(* PLC project VGP - Station 1, CCRE VGP 1.0 *)
(* stored: creationDateTime 2016-05-18T12:27:41, modificationDateTime 2020-06-25T10:53:04 *)

FUNCTION Convert_Pressure : BOOL
  VAR_INPUT
    rawPressure : INT;
  END_VAR
  VAR_OUTPUT
    finalPressure : REAL;
  END_VAR

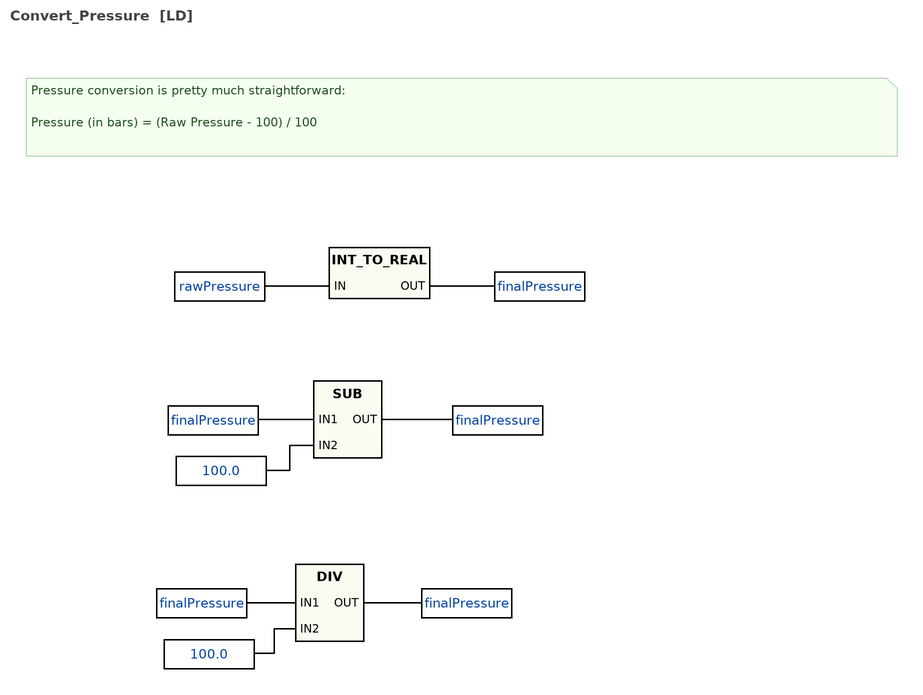
(* LD diagram, written out as Structured Text *)
(* Pressure conversion is pretty much straightforward:

Pressure (in bars) = (Raw Pressure - 100) / 100 *)
finalPressure := INT_TO_REAL(rawPressure);
finalPressure := finalPressure - 100.0;
finalPressure := finalPressure / 100.0;
END_FUNCTION

FUNCTION Finish_Intermediate_Mode : BOOL
  VAR_INPUT
    flow_rate1 : INT;
    flow_rate2 : INT;
    flow_limit : INT;
  END_VAR
  VAR
    negative_flow_limit : INT;
  END_VAR
  VAR_OUTPUT
    Q : BOOL;
  END_VAR

negative_flow_limit := 0 - flow_limit;

IF (negative_flow_limit < flow_rate1) AND (flow_rate1 < flow_limit) THEN
  IF (negative_flow_limit < flow_rate2) AND (flow_rate2 < flow_limit) THEN
    Q := TRUE;
  ELSE
    Q := FALSE;
  END_IF;
ELSE
  Q := FALSE;
END_IF;
          
END_FUNCTION

FUNCTION_BLOCK Verify_Mode_Change
  VAR_INPUT
    mode : INT;
  END_VAR
  VAR_OUTPUT
    Q : BOOL;
  END_VAR
  VAR
    previous_mode : INT := 0;
  END_VAR

IF mode <> previous_mode THEN
  IF (mode > 0) AND (previous_mode > 0) THEN
    Q := TRUE;
  ELSE
    Q := FALSE;
  END_IF;
ELSE
  Q := FALSE;
END_IF;

previous_mode := mode;
          
END_FUNCTION_BLOCK

PROGRAM VGP
  VAR
    raw_pressure AT %IW0 : INT;  (* MODBUS Input Register Address 0 - Pressure as seen from the sensor *)
    raw_tank_lvl AT %IW1 : INT;  (* MODBUS Input Register Address 1 - Tank level as seen from the sensor *)
    raw_dispatch_flow AT %IW2 : INT;  (* MODBUS Input Register Address 2 - Flow rate on the dispatch valve as seen from the sensor *)
    raw_returnline_flow AT %IW3 : INT;  (* MODBUS Input Register Address 3 - Flow rate on the return line as seen from the sensor *)
    raw_relief_valve_flow AT %IW4 : INT;  (* MODBUS Input Register Address 4 - Flow rate on the relief valve as seen from the sensor *)
    raw_min_sp AT %QW1 : INT;  (* MODBUS Holding Register Address 1 - Minimum setpoint (as integer, withouth conversion) *)
    raw_max_sp AT %QW2 : INT;  (* MODBUS Holding Register Address 2 - Maximum setpoint (as integer, withouth conversion) *)
    operation_mode AT %QW3 : INT;  (* MODBUS Holding Register Address 3 - Operation mode, set by the HMI *)
    manual_pump AT %QW4 : INT;  (* MODBUS Holding Register Address 4 - Toggle pump in manual mode *)
    manual_relief_valve AT %QW5 : INT;  (* MODBUS Holding Register Address 5 - Toggle relief valve in manual mode *)
    manual_dispatch_valve AT %QW6 : INT;  (* MODBUS Holding Register Address 6 - Toggle dispatch valve in manual mode *)
    manual_return_valve AT %QW7 : INT;  (* MODBUS Holding Register Address 7 - Toggle return valve in manual mode *)
    source_tank_flow AT %QW20 : INT;  (* MODBUS Holding Register Address 20 - Source Tank flow rate in KL/h *)
    destination_tank_flow AT %QW21 : INT;  (* MODBUS Holding Register Address 21 - Destination Tank flow rate in KL/h *)
    pump AT %QX0.0 : BOOL;
    dispatch_valve AT %QX0.2 : BOOL;
    return_valve AT %QX0.3 : BOOL;
    relief_valve AT %QX0.1 : BOOL;
  END_VAR
  VAR
    pressure : REAL;
    min_sp : REAL;
    max_sp : REAL;
    recirc_mode : BOOL;
    recirc_dispatch_valve : BOOL;
    recirc_return_valve : BOOL;
    recirc_relief_valve : BOOL;
    recirc_pump : BOOL;
    cargo_mode : BOOL;
    cargo_dispatch_valve : BOOL;
    cargo_return_valve : BOOL;
    cargo_relief_valve : BOOL;
    cargo_pump : BOOL;
    man_mode : BOOL;
    man_dispatch_valve : BOOL;
    man_return_valve : BOOL;
    man_relief_valve : BOOL;
    man_pump : BOOL;
    intermediate_mode : BOOL;
    intermediate_dispatch_valve : BOOL;
    intermediate_return_valve : BOOL;
    intermediate_relief_valve : BOOL;
    intermediate_pump : BOOL;
    TOF0 : TOF;
    mode_change : Verify_Mode_Change;
    T0 : TON;
  END_VAR
  VAR  (* added by the conversion: wires and edge detectors of the diagram *)
    _Convert_Pressure152_finalPressure : ANY;
    _Convert_Pressure152_OUT : BOOL;
    _Convert_Pressure153_finalPressure : ANY;
    _Convert_Pressure153_OUT : BOOL;
    _Convert_Pressure154_finalPressure : ANY;
    _Convert_Pressure154_OUT : BOOL;
    _Finish_Intermediate_Mode215_Q : ANY;
    _Finish_Intermediate_Mode215_OUT : BOOL;
    _LE164_ENO : BOOL;
    _LE164_OUT : BOOL;
    _GE169_ENO : BOOL;
    _GE169_OUT : BOOL;
    _GE173_ENO : BOOL;
    _GE173_OUT : BOOL;
    _LE33_ENO : BOOL;
    _LE33_OUT : BOOL;
    _GE38_ENO : BOOL;
    _GE38_OUT : BOOL;
    _EQ42_OUT : BOOL;
    _EQ183_ENO : BOOL;
    _EQ183_OUT : BOOL;
    _EQ49_ENO : BOOL;
    _EQ49_OUT : BOOL;
    _EQ56_ENO : BOOL;
    _EQ56_OUT : BOOL;
    _EQ63_ENO : BOOL;
    _EQ63_OUT : BOOL;
  END_VAR

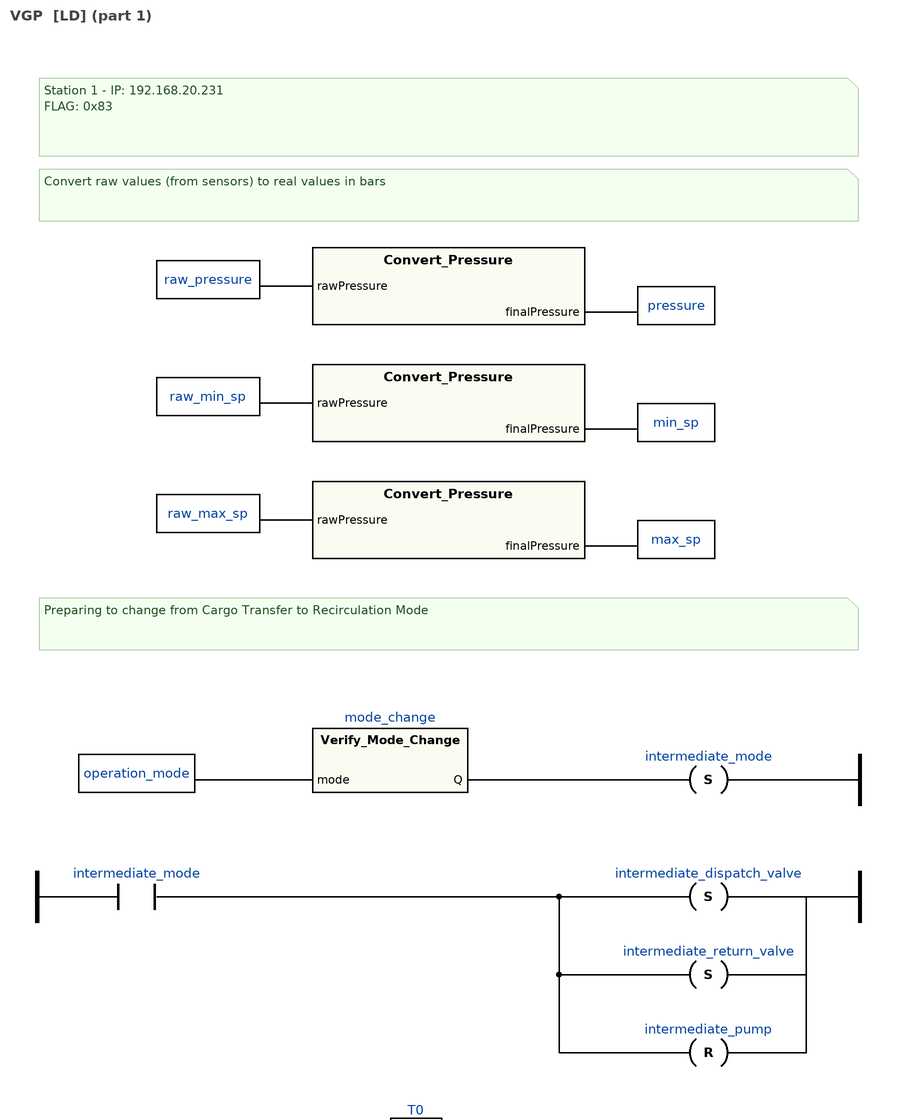
(* LD diagram, written out as Structured Text *)
(* Station 1 - IP: 192.168.20.231
FLAG: 0x83 *)
(* Convert raw values (from sensors) to real values in bars *)
_Convert_Pressure152_OUT := Convert_Pressure(rawPressure := raw_pressure, finalPressure => _Convert_Pressure152_finalPressure);
pressure := _Convert_Pressure152_finalPressure;
_Convert_Pressure153_OUT := Convert_Pressure(rawPressure := raw_min_sp, finalPressure => _Convert_Pressure153_finalPressure);
min_sp := _Convert_Pressure153_finalPressure;
_Convert_Pressure154_OUT := Convert_Pressure(rawPressure := raw_max_sp, finalPressure => _Convert_Pressure154_finalPressure);
max_sp := _Convert_Pressure154_finalPressure;
(* Preparing to change from Cargo Transfer to Recirculation Mode *)
mode_change(mode := operation_mode);
IF mode_change.Q THEN intermediate_mode := TRUE; END_IF;
IF intermediate_mode THEN intermediate_dispatch_valve := TRUE; END_IF;
IF intermediate_mode THEN intermediate_return_valve := TRUE; END_IF;
IF intermediate_mode THEN intermediate_pump := FALSE; END_IF;
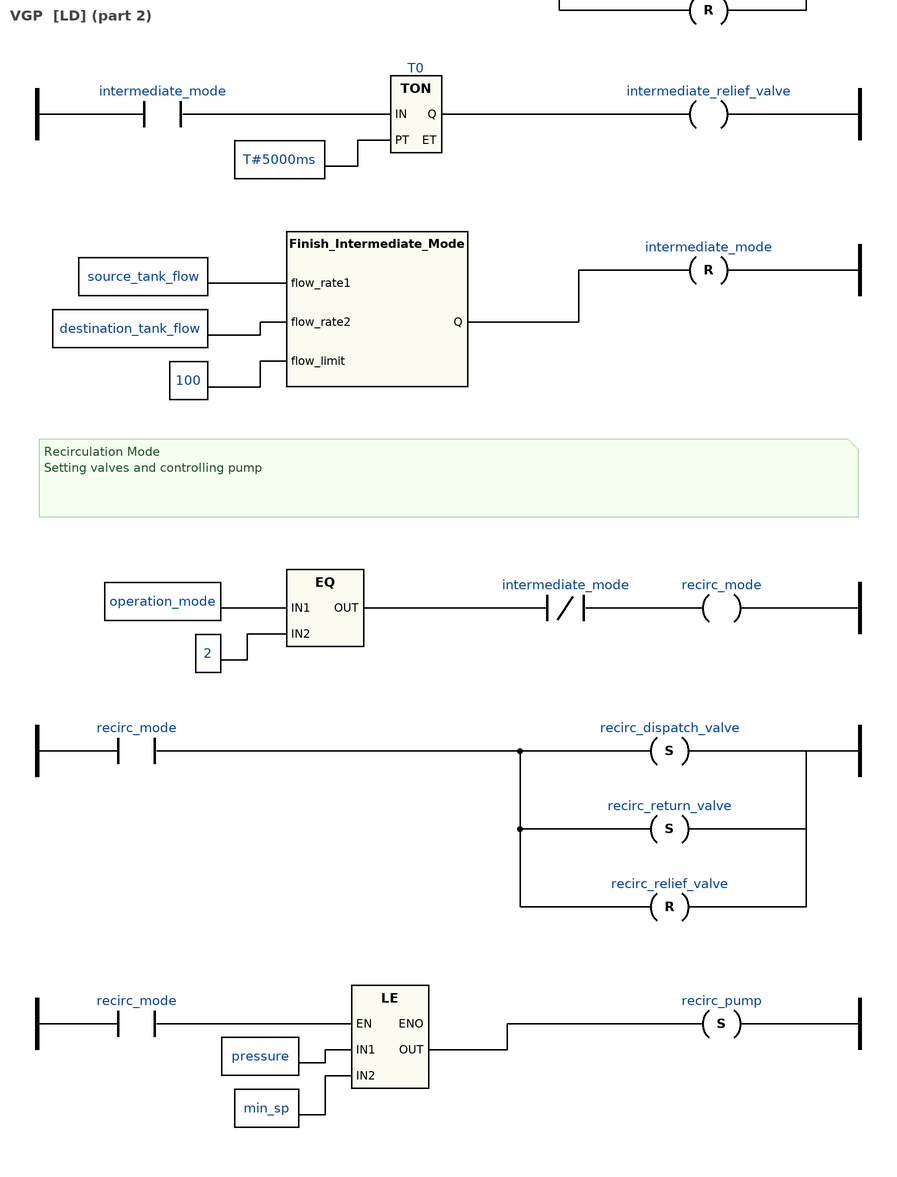
T0(IN := intermediate_mode, PT := T#5000ms);
intermediate_relief_valve := T0.Q;
_Finish_Intermediate_Mode215_OUT := Finish_Intermediate_Mode(flow_rate1 := source_tank_flow, flow_rate2 := destination_tank_flow, flow_limit := 100, Q => _Finish_Intermediate_Mode215_Q);
IF _Finish_Intermediate_Mode215_Q THEN intermediate_mode := FALSE; END_IF;
(* Recirculation Mode
Setting valves and controlling pump *)
recirc_mode := operation_mode = 2 AND NOT intermediate_mode;
IF recirc_mode THEN recirc_dispatch_valve := TRUE; END_IF;
IF recirc_mode THEN recirc_return_valve := TRUE; END_IF;
IF recirc_mode THEN recirc_relief_valve := FALSE; END_IF;
_LE164_OUT := LE(EN := recirc_mode, IN1 := pressure, IN2 := min_sp, ENO => _LE164_ENO);
IF _LE164_OUT THEN recirc_pump := TRUE; END_IF;
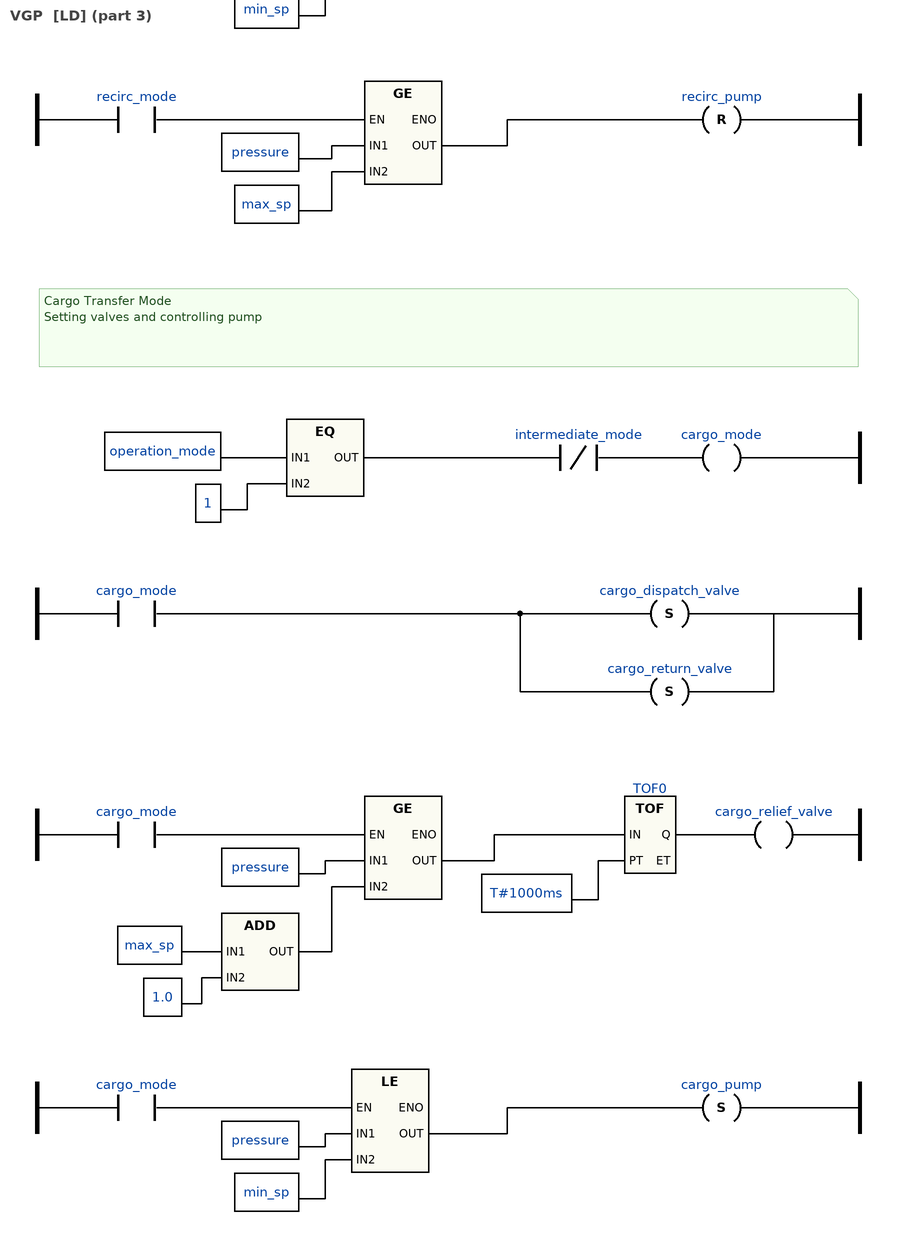
_GE169_OUT := GE(EN := recirc_mode, IN1 := pressure, IN2 := max_sp, ENO => _GE169_ENO);
IF _GE169_OUT THEN recirc_pump := FALSE; END_IF;
(* Cargo Transfer Mode
Setting valves and controlling pump *)
cargo_mode := operation_mode = 1 AND NOT intermediate_mode;
IF cargo_mode THEN cargo_dispatch_valve := TRUE; END_IF;
IF cargo_mode THEN cargo_return_valve := TRUE; END_IF;
_GE173_OUT := GE(EN := cargo_mode, IN1 := pressure, IN2 := max_sp + 1.0, ENO => _GE173_ENO);
TOF0(IN := _GE173_OUT, PT := T#1000ms);
cargo_relief_valve := TOF0.Q;
_LE33_OUT := LE(EN := cargo_mode, IN1 := pressure, IN2 := min_sp, ENO => _LE33_ENO);
IF _LE33_OUT THEN cargo_pump := TRUE; END_IF;
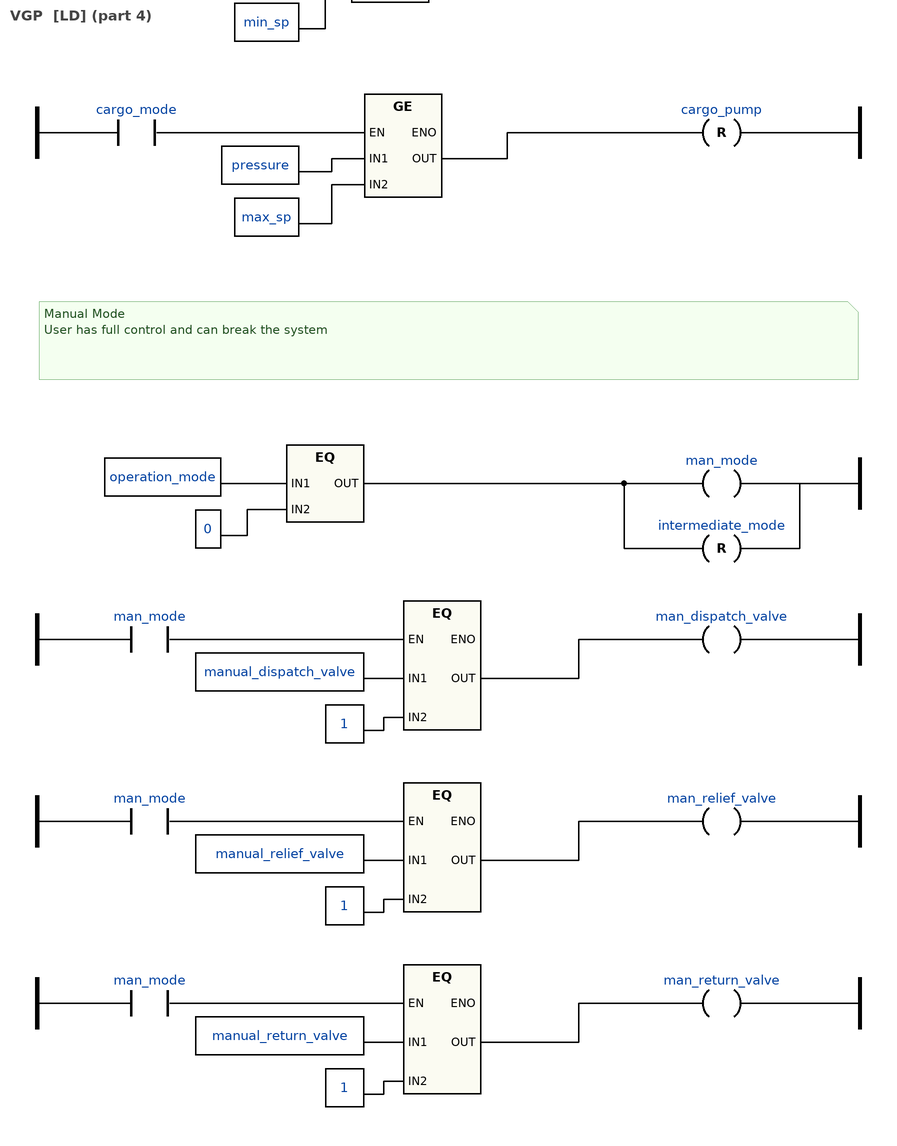
_GE38_OUT := GE(EN := cargo_mode, IN1 := pressure, IN2 := max_sp, ENO => _GE38_ENO);
IF _GE38_OUT THEN cargo_pump := FALSE; END_IF;
(* Manual Mode
User has full control and can break the system *)
_EQ42_OUT := operation_mode = 0;
man_mode := _EQ42_OUT;
IF _EQ42_OUT THEN intermediate_mode := FALSE; END_IF;
_EQ183_OUT := EQ(EN := man_mode, IN1 := manual_dispatch_valve, IN2 := 1, ENO => _EQ183_ENO);
man_dispatch_valve := _EQ183_OUT;
_EQ49_OUT := EQ(EN := man_mode, IN1 := manual_relief_valve, IN2 := 1, ENO => _EQ49_ENO);
man_relief_valve := _EQ49_OUT;
_EQ56_OUT := EQ(EN := man_mode, IN1 := manual_return_valve, IN2 := 1, ENO => _EQ56_ENO);
man_return_valve := _EQ56_OUT;
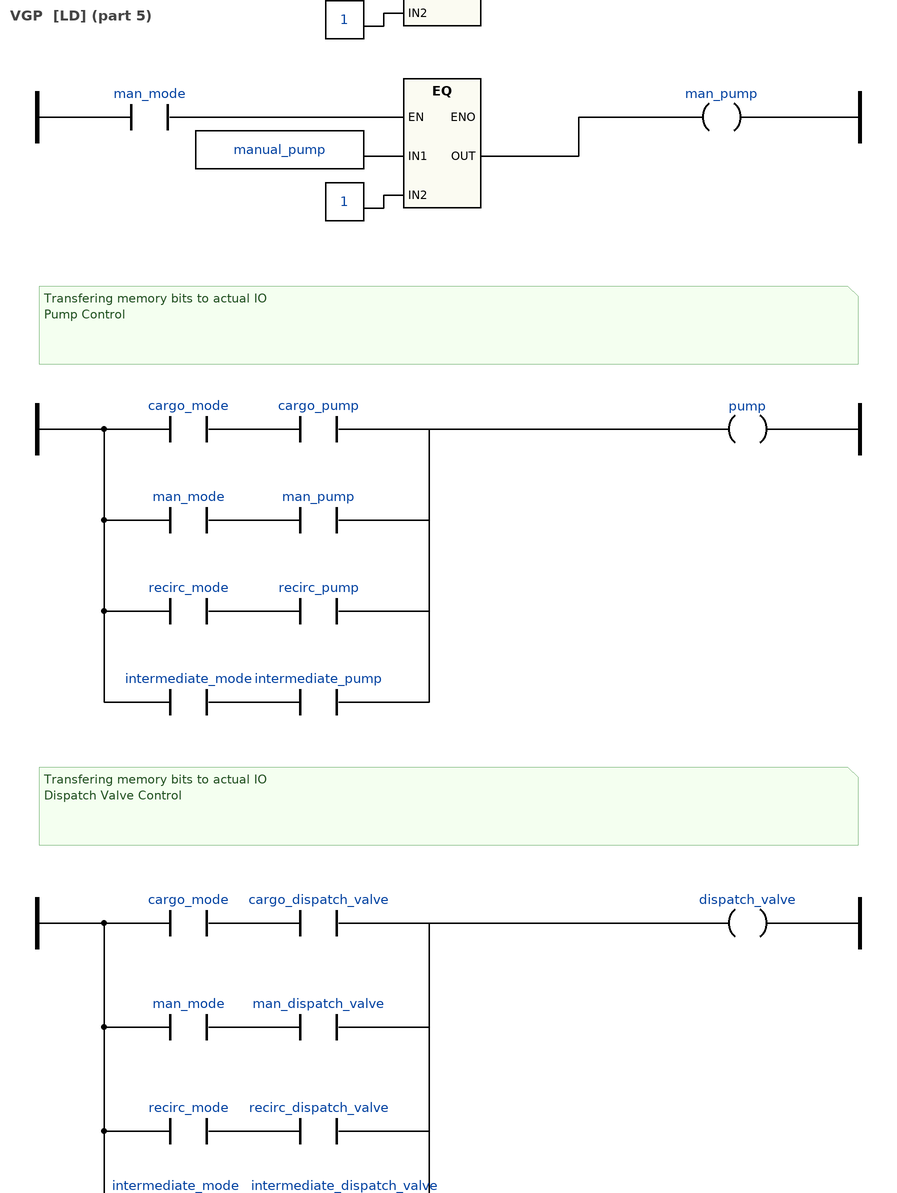
_EQ63_OUT := EQ(EN := man_mode, IN1 := manual_pump, IN2 := 1, ENO => _EQ63_ENO);
man_pump := _EQ63_OUT;
(* Transfering memory bits to actual IO
Pump Control *)
pump := cargo_mode AND cargo_pump OR man_mode AND man_pump OR recirc_mode AND recirc_pump OR intermediate_mode AND intermediate_pump;
(* Transfering memory bits to actual IO
Dispatch Valve Control *)
dispatch_valve := cargo_mode AND cargo_dispatch_valve OR man_mode AND man_dispatch_valve OR recirc_mode AND recirc_dispatch_valve OR intermediate_mode AND intermediate_dispatch_valve;
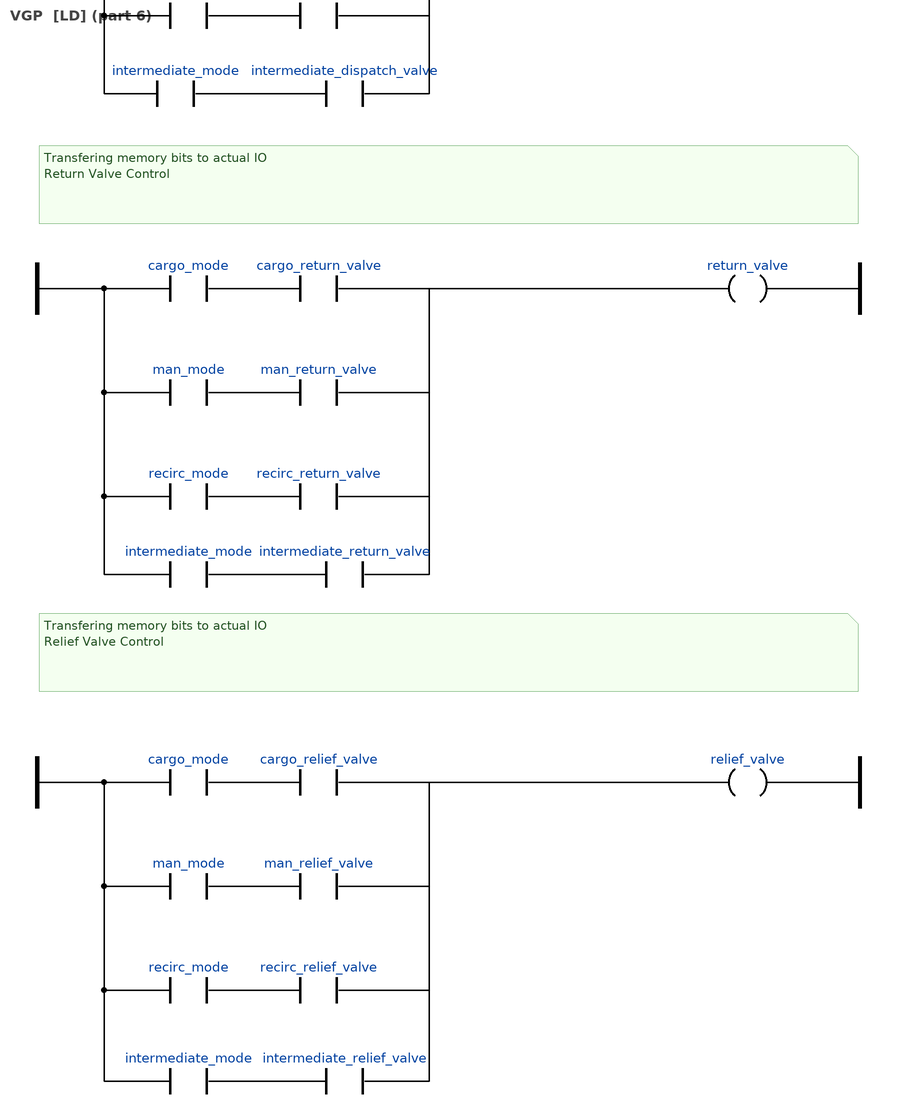
(* Transfering memory bits to actual IO
Return Valve Control *)
return_valve := cargo_mode AND cargo_return_valve OR man_mode AND man_return_valve OR recirc_mode AND recirc_return_valve OR intermediate_mode AND intermediate_return_valve;
(* Transfering memory bits to actual IO
Relief Valve Control *)
relief_valve := cargo_mode AND cargo_relief_valve OR man_mode AND man_relief_valve OR recirc_mode AND recirc_relief_valve OR intermediate_mode AND intermediate_relief_valve;
END_PROGRAM

CONFIGURATION Config0
  RESOURCE Res0 ON PLC
    TASK TaskMain(INTERVAL := T#50ms, PRIORITY := 0);
    PROGRAM Inst0 WITH TaskMain : VGP;
  END_RESOURCE
END_CONFIGURATION
